{attribute 'GeneratedUsingTerminal: EL3351-0000-0016'}
{attribute addProperty BoxType "EL3351-0000-0016"}
{attribute addProperty Id "AIBridge_InputsAT %I*AIBridge_Inputs_555AA1E89AISupply_InputsAT %I*AISupply_Inputs_555AA1E89WcStateAT %I*WcState_9091E0EB2InfoDataAT %I*InfoData_94A18F5E2"}
{attribute addProperty CRC "930421242"}
{attribute addProperty Size "22"}
TYPE EL3351_377519FA EXTENDS EtcSlaveTerminalBase_947E5A46 :
STRUCT
	{attribute addProperty Name "AIBridge_Inputs"}
	AIBridge_Inputs : AIBridge_Inputs_555AA1E8;
	{attribute addProperty Name "AISupply_Inputs"}
	AISupply_Inputs : AISupply_Inputs_555AA1E8;
	{attribute addProperty Name "WcState"}
	WcState : WcState_9091E0EB;
	{attribute addProperty Name "InfoData"}
	InfoData : InfoData_94A18F5E;
END_STRUCT
END_TYPE

(* stored: Version 1.2.0.0, ProductVersion 3.1.4024.9
   DUT EL3351_377519FA: Id {960e7bab-f7d4-4485-a578-0fb469bedf2c} *)
